{attribute addProperty BoxType "EL3114-0000-0016"}
{attribute addProperty Id "AI_Standard_ChannelAT %I*ARRAY[0..6] OF AI_Standard_Channel_8749C235296370WcStateAT %I*WcState_98A4DF7520.250InfoDataAT %I*InfoData_BC63D37F80100"}
{attribute addProperty CRC "2617007306"}
{attribute addProperty SizeInBites "378"}
{attribute addProperty SizeInBytes "47.25"}
TYPE EL3114_8F040432 :
STRUCT
	{attribute addProperty Name "AI_Standard_Channel"}
	AI_Standard_Channel : ARRAY[0..6] OF AI_Standard_Channel_8749C235;
	{attribute addProperty Name "WcState"}
	WcState : WcState_98A4DF75;
	{attribute addProperty Name "InfoData"}
	InfoData : InfoData_BC63D37F;
END_STRUCT
END_TYPE

(* stored: Version 1.2.0.0, ProductVersion 3.1.4024.9
   DUT EL3114_8F040432: Id {4429c135-64f6-463a-b1b4-35f21e707c8c} *)
